{attribute 'qualified_only'}
{attribute 'strict'}
{attribute 'to_string'}
TYPE E_SeqMOVITRAC_B_WithBrake :
(
	INIT := 0,
	STOPPED,
	RELEASE_BRAKE,
	MOVING_FORWARD,
	MOVING_BACKWARD,
	STOPPING,
	APPLY_BRAKE,
	ERROR
);
END_TYPE

(* stored: Version 1.1.0.1, ProductVersion 3.1.4024.12
   DUT E_SeqMOVITRAC_B_WithBrake: Id {a16bc342-e72f-4c40-a27e-a793ea358007} *)
